SUBAPPLICATION Uebung_172_ASRT (* Exercise for ASRT_AX_T_FF_SR *)
  (* Standard: 61499-2; Description: Copyright (c) 2026 Meisterschulen am Ostbahnhof This program and the accompanying materials are made available under the terms of the Eclipse Public License 2.0 which is available at https://www.eclipse.org/legal/epl-2.0/ SPDX-License-Identifier: EPL-2.0 *)
  (* Version 1.0, 2026-09-03, Franz Höpfinger, Meisterschulen am Ostbahnhof, initial API and implementation and/or initial documentation *)
  PACKAGE Uebungen;
  IMPORT logiBUS::io::DI::logiBUS_DI::Input_I1;
  IMPORT logiBUS::io::DI::logiBUS_DI::Input_I2;
  IMPORT logiBUS::io::DI::logiBUS_DI::Input_I3;
  IMPORT logiBUS::io::DI::logiBUS_DI_Events::BUTTON_SINGLE_CLICK;
  IMPORT logiBUS::io::DQ::logiBUS_DO::Output_Q1;
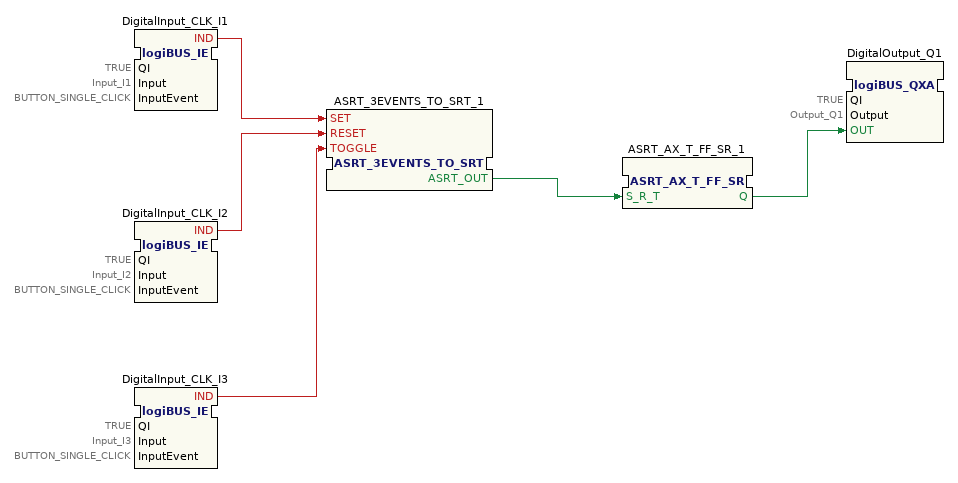
  FBS
    ASRT_AX_T_FF_SR_1 : adapter::events::unidirectional::ASRT_AX_T_FF_SR;
    ASRT_3EVENTS_TO_SRT_1 : adapter::conversion::unidirectional::ASRT_3EVENTS_TO_SRT;
    DigitalInput_CLK_I1 : logiBUS::io::DI::logiBUS_IE(QI := TRUE, Input := Input_I1, InputEvent := BUTTON_SINGLE_CLICK);
    DigitalOutput_Q1 : logiBUS::io::DQ::logiBUS_QXA(QI := TRUE, Output := Output_Q1);
    DigitalInput_CLK_I2 : logiBUS::io::DI::logiBUS_IE(QI := TRUE, Input := Input_I2, InputEvent := BUTTON_SINGLE_CLICK);
    DigitalInput_CLK_I3 : logiBUS::io::DI::logiBUS_IE(QI := TRUE, Input := Input_I3, InputEvent := BUTTON_SINGLE_CLICK);
  END_FBS
  EVENT_CONNECTIONS
    DigitalInput_CLK_I1.IND TO ASRT_3EVENTS_TO_SRT_1.SET;
    DigitalInput_CLK_I2.IND TO ASRT_3EVENTS_TO_SRT_1.RESET;
    DigitalInput_CLK_I3.IND TO ASRT_3EVENTS_TO_SRT_1.TOGGLE;
  END_CONNECTIONS
  ADAPTER_CONNECTIONS
    ASRT_3EVENTS_TO_SRT_1.ASRT_OUT TO ASRT_AX_T_FF_SR_1.S_R_T;
    ASRT_AX_T_FF_SR_1.Q TO DigitalOutput_Q1.OUT;
  END_CONNECTIONS
END_SUBAPPLICATION
